// TwinCAT 3 PLC project EXERCISES
// ProgramVersion: 3.1.4023.0
// libraries:
//   CmpBitmapPool, * (System)
//   Tc2_Standard, * (Beckhoff Automation GmbH)
//   Tc2_System, * (Beckhoff Automation GmbH)
//   Tc3_Module, * (Beckhoff Automation GmbH)
// project tree:
//   / GlobalTextList.TcGTLO, PlcTask.TcTTO, Visualization Manager.TcVMO (not stored)
//   POUs/ ImagePool.TcIPO (not stored), MAIN.TcPOU, Knipperlicht.TcPOU, Verkeerslicht.TcPOU, Verkeerslicht_Multiple.TcPOU
//   VISUs/ Verkeerslicht_Multiple.TcVIS
// real-time tasks:
//   TASK PlcTask: cycle T#10ms, priority 20, ADS port 350

CONFIGURATION EXERCISES
    RESOURCE PLC ON TwinCAT3
        TASK PlcTask(INTERVAL := T#10ms, PRIORITY := 20);
        PROGRAM MAIN WITH PlcTask : MAIN;
    END_RESOURCE
END_CONFIGURATION

// ---- POUs/MAIN.TcPOU
PROGRAM MAIN
VAR
END_VAR

Verkeerslicht_Multiple();

END_PROGRAM

// ---- POUs/Verkeerslicht_Multiple.TcPOU
PROGRAM Verkeerslicht_Multiple

VAR_INPUT
	S_P_H : BOOL;
	S_P_V : BOOL;
END_VAR

VAR_OUTPUT
	// Horizontal
	LED_H_G : BOOL;
	LED_H_Y : BOOL;
	LED_H_R : BOOL;
	
	LED_P_H_G : BOOL;
	LED_P_H_R : BOOL;
	
	// Vertical
	LED_V_G : BOOL;
	LED_V_Y : BOOL;
	LED_V_R : BOOL;

	LED_P_V_G : BOOL;
	LED_P_V_R : BOOL;
END_VAR

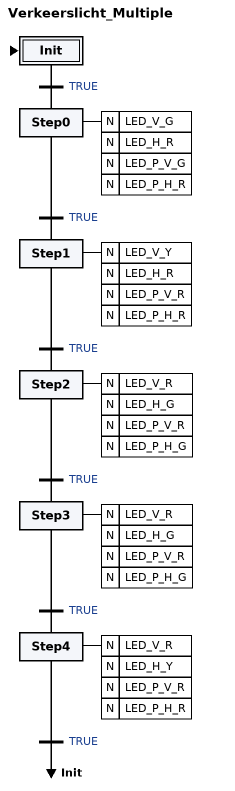
INITIAL_STEP Init:
END_STEP
TRANSITION FROM Init TO Step0
    := TRUE;
END_TRANSITION
STEP Step0:  // min time T#10s, max time T#20s
    LED_V_G(N);
    LED_H_R(N);
    LED_P_V_G(N);
    LED_P_H_R(N);
END_STEP
TRANSITION FROM Step0 TO Step1
    := TRUE;
END_TRANSITION
STEP Step1:  // min time T#5s
    LED_V_Y(N);
    LED_H_R(N);
    LED_P_V_R(N);
    LED_P_H_R(N);
END_STEP
TRANSITION FROM Step1 TO Step2
    := TRUE;
END_TRANSITION
STEP Step2:  // min time T#15s
    LED_V_R(N);
    LED_H_G(N);
    LED_P_V_R(N);
    LED_P_H_G(N);
END_STEP
TRANSITION FROM Step2 TO Step3
    := TRUE;
END_TRANSITION
STEP Step3:  // min time T#5s
    LED_V_R(N);
    LED_H_G(N);
    LED_P_V_R(N);
    LED_P_H_G(N);
END_STEP
TRANSITION FROM Step3 TO Step4
    := TRUE;
END_TRANSITION
STEP Step4:  // min time T#5s
    LED_V_R(N);
    LED_H_Y(N);
    LED_P_V_R(N);
    LED_P_H_R(N);
END_STEP
TRANSITION FROM Step4 TO Init
    := TRUE;
END_TRANSITION

END_PROGRAM

// ---- POUs/Knipperlicht.TcPOU
PROGRAM Knipperlicht
VAR_INPUT
	S01: BOOL;
END_VAR
VAR_OUTPUT
	Q01: BOOL;
END_VAR
VAR
END_VAR

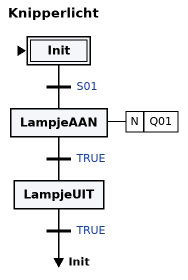
INITIAL_STEP Init:
END_STEP
TRANSITION FROM Init TO LampjeAAN
    := S01;
END_TRANSITION
STEP LampjeAAN:  // min time T#700ms
    Q01(N);
END_STEP
TRANSITION FROM LampjeAAN TO LampjeUIT
    := TRUE;
END_TRANSITION
STEP LampjeUIT:  // min time T#300ms
END_STEP
TRANSITION FROM LampjeUIT TO Init
    := TRUE;
END_TRANSITION

END_PROGRAM

// ---- POUs/Verkeerslicht.TcPOU
PROGRAM Verkeerslicht
VAR
END_VAR

VAR_OUTPUT
	LED_V_G : BOOL;
	LED_V_Y : BOOL;
	LED_V_R : BOOL;

	LED_H_G : BOOL;
	LED_H_Y : BOOL;
	LED_H_R : BOOL;
END_VAR

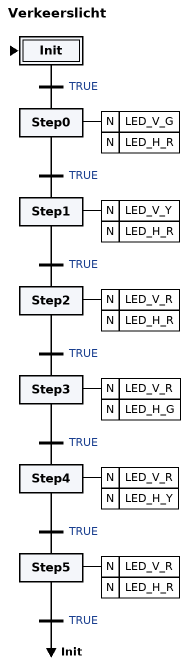
INITIAL_STEP Init:
END_STEP
TRANSITION FROM Init TO Step0
    := TRUE;
END_TRANSITION
STEP Step0:  // min time T#20s
    LED_V_G(N);
    LED_H_R(N);
END_STEP
TRANSITION FROM Step0 TO Step1
    := TRUE;
END_TRANSITION
STEP Step1:  // min time T#5s
    LED_V_Y(N);
    LED_H_R(N);
END_STEP
TRANSITION FROM Step1 TO Step2
    := TRUE;
END_TRANSITION
STEP Step2:  // min time T#5s
    LED_V_R(N);
    LED_H_R(N);
END_STEP
TRANSITION FROM Step2 TO Step3
    := TRUE;
END_TRANSITION
STEP Step3:  // min time T#20s
    LED_V_R(N);
    LED_H_G(N);
END_STEP
TRANSITION FROM Step3 TO Step4
    := TRUE;
END_TRANSITION
STEP Step4:  // min time T#5s
    LED_V_R(N);
    LED_H_Y(N);
END_STEP
TRANSITION FROM Step4 TO Step5
    := TRUE;
END_TRANSITION
STEP Step5:  // min time T#5s
    LED_V_R(N);
    LED_H_R(N);
END_STEP
TRANSITION FROM Step5 TO Init
    := TRUE;
END_TRANSITION

END_PROGRAM

// ---- VISUs/Verkeerslicht_Multiple.TcVIS
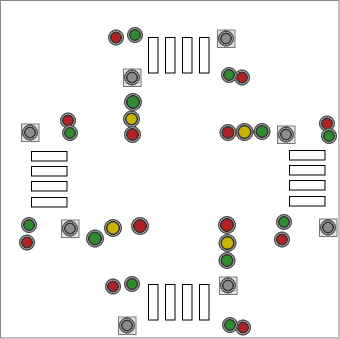
VISUALIZATION Verkeerslicht_Multiple  // 340x339, background image ImagePool.Verkeerslicht_01
    Lamp1 (122,125 21x19), variable: Verkeerslicht_Multiple.LED_V_R, style: Lamp-Lamp1-Red
    Lamp1 (122,109 19x20), variable: Verkeerslicht_Multiple.LED_V_Y, style: Lamp-Lamp1-Yellow
    Lamp1 (122,92 22x20), variable: Verkeerslicht_Multiple.LED_V_G, style: Lamp-Lamp1-Green
    Lamp1 (217,215 20x20), variable: Verkeerslicht_Multiple.LED_V_R, style: Lamp-Lamp1-Red
    Lamp1 (217,233 21x20), variable: Verkeerslicht_Multiple.LED_V_Y, style: Lamp-Lamp1-Yellow
    Lamp1 (217,251 20x19), variable: Verkeerslicht_Multiple.LED_V_G, style: Lamp-Lamp1-Green
    Lamp1 (121,216 38x20), variable: Verkeerslicht_Multiple.LED_H_R, style: Lamp-Lamp1-Red
    Lamp1 (103,216 20x24), variable: Verkeerslicht_Multiple.LED_H_Y, style: Lamp-Lamp1-Yellow
    Lamp1 (85,216 20x45), variable: Verkeerslicht_Multiple.LED_H_G, style: Lamp-Lamp1-Green
    Lamp1 (217,123 22x19), variable: Verkeerslicht_Multiple.LED_H_R, style: Lamp-Lamp1-Red
    Lamp1 (234,122 21x20), variable: Verkeerslicht_Multiple.LED_H_Y, style: Lamp-Lamp1-Yellow
    Lamp1 (251,122 22x19), variable: Verkeerslicht_Multiple.LED_H_G, style: Lamp-Lamp1-Green
    Rectangle (31,151 36x10)
    Rectangle (31,166 36x10)
    Rectangle (31,181 36x10)
    Rectangle (31,197 36x10)
    Rectangle (289,150 36x10)
    Rectangle (289,165 36x10)
    Rectangle (289,180 36x10)
    Rectangle (289,196 36x10)
    Rectangle (169,50 36x10), angle 90
    Rectangle (152,50 36x10), angle 90
    Rectangle (186,50 36x10), angle 90
    Rectangle (135,50 36x10), angle 90
    Rectangle (169,297 36x10), angle 90
    Rectangle (152,297 36x10), angle 90
    Rectangle (186,297 36x10), angle 90
    Rectangle (135,297 36x10), angle 90
    PushSwitch (61,217 18x23), variable: VerkeersLicht_2.S01, behaviour: TOGGLE, style: Switch-PushSwitch-Gray
    PushSwitch (21,121 18x23), variable: VerkeersLicht_2.S01, behaviour: TOGGLE, style: Switch-PushSwitch-Gray
    PushSwitch (118,314 18x23), variable: VerkeersLicht_2.S02, behaviour: TOGGLE, style: Switch-PushSwitch-Gray
    PushSwitch (219,274 18x23), variable: VerkeersLicht_2.S02, behaviour: TOGGLE, style: Switch-PushSwitch-Gray
    PushSwitch (319,216 18x23), variable: VerkeersLicht_2.S01, behaviour: TOGGLE, style: Switch-PushSwitch-Gray
    PushSwitch (277,123 18x23), variable: VerkeersLicht_2.S01, behaviour: TOGGLE, style: Switch-PushSwitch-Gray
    PushSwitch (123,66 18x23), variable: VerkeersLicht_2.S02, behaviour: TOGGLE, style: Switch-PushSwitch-Gray
    PushSwitch (217,27 18x23), variable: VerkeersLicht_2.S02, behaviour: TOGGLE, style: Switch-PushSwitch-Gray
    Lamp1 (18,231 18x23), variable: Verkeerslicht_Multiple.LED_P_V_R, style: Lamp-Lamp1-Red
    Lamp1 (18,216 22x18), variable: Verkeerslicht_Multiple.LED_P_V_G, style: Lamp-Lamp1-Green
    Lamp1 (59,109 18x23), variable: Verkeerslicht_Multiple.LED_P_V_R, style: Lamp-Lamp1-Red
    Lamp1 (59,124 22x18), variable: Verkeerslicht_Multiple.LED_P_V_G, style: Lamp-Lamp1-Green
    Lamp1 (273,228 18x23), variable: Verkeerslicht_Multiple.LED_P_V_R, style: Lamp-Lamp1-Red
    Lamp1 (273,213 22x18), variable: Verkeerslicht_Multiple.LED_P_V_G, style: Lamp-Lamp1-Green
    Lamp1 (107,26 18x23), variable: Verkeerslicht_Multiple.LED_P_H_R, style: Lamp-Lamp1-Red
    Lamp1 (124,26 22x18), variable: Verkeerslicht_Multiple.LED_P_H_G, style: Lamp-Lamp1-Green
    Lamp1 (318,112 18x23), variable: Verkeerslicht_Multiple.LED_P_V_R, style: Lamp-Lamp1-Red
    Lamp1 (318,127 22x18), variable: Verkeerslicht_Multiple.LED_P_V_G, style: Lamp-Lamp1-Green
    Lamp1 (104,275 18x23), variable: Verkeerslicht_Multiple.LED_P_H_R, style: Lamp-Lamp1-Red
    Lamp1 (121,275 22x18), variable: Verkeerslicht_Multiple.LED_P_H_G, style: Lamp-Lamp1-Green
    Lamp1 (233,66 18x23), variable: Verkeerslicht_Multiple.LED_P_H_R, style: Lamp-Lamp1-Red
    Lamp1 (218,66 22x18), variable: Verkeerslicht_Multiple.LED_P_H_G, style: Lamp-Lamp1-Green
    Lamp1 (234,316 18x23), variable: Verkeerslicht_Multiple.LED_P_H_R, style: Lamp-Lamp1-Red
    Lamp1 (219,316 22x18), variable: Verkeerslicht_Multiple.LED_P_H_G, style: Lamp-Lamp1-Green
END_VISUALIZATION
